INTERFACE PUBLIC FilterDifferentialPressureProvider EXTENDS __System.IQueryInterface

PROPERTY PUBLIC Pressure : LREAL
GET
END_GET
END_PROPERTY

END_INTERFACE

(* stored: Version 1.1.0.1, ProductVersion 3.1.4026.18
   Itf FilterDifferentialPressureProvider: Id {28206f5b-98c3-4ddf-850e-79df68a91151}
   Property Pressure: Id {7cca8b22-a4e3-4ee4-b46a-a7d791cd1b34}
   Get Get: Id {1a4f04aa-c518-496d-b9c2-9846bbc509a1} *)
